{attribute 'GeneratedUsingTerminal: EK1100-0000-0018'}
{attribute addProperty BoxType "EK1100-0000-0018"}
{attribute addProperty Id "TcTerminals210_2BK1250TcTerminals210_2BK1250_CEF741550"}
{attribute addProperty CRC "1354842929"}
{attribute addProperty Size "0"}
TYPE TcTerminals210_EK1100_2_50C14331 EXTENDS EK1100_1FC0878B :
STRUCT
	{attribute addProperty Name "TcTerminals210_2BK1250"}
	{attribute addProperty PreviousPort "TcTerminals210_EK1100_2 : B"}
	TcTerminals210_2BK1250 : TcTerminals210_2BK1250_CEF74155;
END_STRUCT
END_TYPE

(* stored: Version 1.2.0.0, ProductVersion 3.1.4024.9
   DUT TcTerminals210_EK1100_2_50C14331: Id {5fb47d0c-0eac-4394-9dd2-9f46b3556b76} *)
